// TIA Portal V19 export
TYPE "LAF_typeEmStatus"
// Status of the equipment module
// stored: Access Published
   STRUCT
      enabled { ExternalWritable := 'False'} : Bool;   // Equipment module is enabled
      acknowledgeActive { ExternalWritable := 'False'} : Bool;   // Acknowledge command active
      alarmsDisabled { ExternalWritable := 'False'} : Bool;   // The alarms of the equipment module are disabled
      simulationActive { ExternalWritable := 'False'} : Bool;   // The simulation of the equipment module is active
      safetyReleased { ExternalWritable := 'False'} : Bool;   // Safety released
      initialized { ExternalWritable := 'False'} : Bool;   // Equipment module is initialized
      homed { ExternalWritable := 'False'} : Bool;   // Equipment module is homed
      safeState { ExternalWritable := 'False'} : Bool;   // Equipment module is in a safe state
      stateComplete { ExternalWritable := 'False'} : Bool;   // Equipment module has completed the current unit status
   END_STRUCT;
END_TYPE
